// TIA Portal V18 export
DATA_BLOCK "magnet__DB"   // DB70
VERSION : 0.1
// stored: AutoNumber true, DBAccessibleFromOPCUA true, InstanceOfName magnet_, InstanceOfType FB
"magnet_"
   // VAR_INPUT
   //    sensor : Bool;
   // END_VAR
   // VAR_OUTPUT
   //    y : Bool;
   // END_VAR
   // VAR
   //    energize : Bool;
   // END_VAR
   // VAR RETAIN
   //    seconds : Real;
   // END_VAR
   // VAR
   //    ton { S7_SetPoint := 'True'} : TON_TIME;
   //    pt_ms : Time;
   // END_VAR
BEGIN
END_DATA_BLOCK
